FUNCTION_BLOCK UN_CleanroomConnect EXTENDS Un_Base
VAR
//------------------------------------------//
//Function Blocks

//------------------------------------------//



//------------------------------------------//
//Control Modules (Devices)
	s_CmKmweLeds 				: CM_KmweLeds;
//------------------------------------------//

//------------------------------------------//
//Inputs
	s_diEmergencyBtn			: FB_DigInput;
//------------------------------------------//

//------------------------------------------//
//Alarms
	s_errEmergencyBtn			: FB_AlarmHandler;
//------------------------------------------//
	
//------------------------------------------//
//Params

//------------------------------------------//

//------------------------------------------//
//Variables
	s_stSqldbSettings			: ST_SqLdbConfiguration;
//------------------------------------------//

//------------------------------------------//
//Properties

//------------------------------------------//

//------------------------------------------//
//Hmi
	s_fbHmiBtnAutomatic			: FB_HmiBtn;
	s_fbHmiBtnManual			: FB_HmiBtn;
	s_fbHmiBtnTesterConfig		: FB_HmiBtn;
	s_fbHmiBtnAlarms			: FB_HmiBtn;
//------------------------------------------//
END_VAR


SUPER^();

METHOD PROTECTED _m_Alarms : BOOL

IF NOT SUPER^._m_Alarms() THEN
	RETURN;
END_IF

//overbruggen in automode tot en met place table blablabla
s_errEmergencyBtn(i_bStaActive 			:= NOT s_DiEmergencyBtn.p_bStaInput AND NOT GVL.g_fbHmiBtnSimulation.p_bStaBtn AND GVL.g_bConnectTestEquipment ,
				  i_eAlarmLevel 		:= E_AlarmLevel.Alarm,
				  i_sAlarmText 			:= 'Emergency button pressed');

IF GVL_KMWEGenericLib.g_fbAlarmManager.p_bAlarmActive THEN 
	GVL.g_eStaLedColor := E_KmweLedColors.Red;
END_IF

s_bStaError := s_errEmergencyBtn.q_bStaActive;

_m_Alarms := TRUE;
END_METHOD

METHOD PROTECTED _m_Devices : BOOL

IF NOT SUPER^._m_Devices() THEN
	RETURN;
END_IF

//------------------------------------------//
//CM
	s_CmKmweLeds(i_bReqEnable := TRUE,
			 i_bCmdReset  := s_bCmdReset,
			 i_eCtrlMode  := s_eCtrlMode,
			 i_eColor 	  := GVL.g_eStaLedColor);
			 
	s_CmKmweLeds.p_bFlashFast := GVL.g_bLedFlashFast;
	s_CmKmweLeds.p_bFlashSlow := GVL.g_bLedFlashSlow;

//------------------------------------------//

//------------------------------------------//
//Outputs
//------------------------------------------//

//------------------------------------------//
//Inputs
	s_diEmergencyBtn();	
//------------------------------------------//

_m_Devices := TRUE;
END_METHOD

METHOD PROTECTED _m_Hmi : BOOL
VAR_INST
	s_sPrevPageAlarms 		: STRING;
	s_sPrevBottom1Alarms	: STRING;
	
	s_sCompanySelectionVisible	: STRING;
END_VAR

IF NOT SUPER^._m_Hmi() THEN
	RETURN;
END_IF

//------------------------------------------//
//Mode management
IF GVL_KMWEGenericLib.g_fbHmiBtnReturnToStart.p_osfBtnPress THEN
	s_eCtrlMode := E_CtrlMode.IDLE;

	GVL_KMWEGenericLib.g_fbHmiBtnAcknowledge.p_bStaVisible	:= TRUE;
	GVL_KMWEGenericLib.g_fbHmiBtnAcknowledge.p_bStaEnabled	:= TRUE;	
END_IF
//------------------------------------------//

//------------------------------------------//
//Alarm Button can always be pressed
IF s_fbHmiBtnAlarms.p_osrBtnPress AND GVL.g_sToHmiMiddleContent <> GVL.g_stHmiMiddle.AlarmManager THEN
	s_sPrevPageAlarms			:= GVL.g_sToHmiMiddleContent;
	s_sPrevBottom1Alarms		:= GvL.g_sToHmiBottomContent;
	GVL.g_sToHmiMiddleContent 	:= GVL.g_stHmiMiddle.AlarmManager;
	GVL.g_sToHmiBottomContent	:= GVL.g_stHmiBottomBar.Alarm;
	
	GVL_KMWEGenericLib.g_fbHmiBtnReturn.p_bStaVisible 			:= TRUE;
	GVL_KMWEGenericLib.g_fbHmiBtnReturn.p_bStaEnabled 			:= TRUE;
END_IF

IF GVL.g_sToHmiMiddleContent = GVL.g_stHmiMiddle.AlarmManager AND GVL_KMWEGenericLib.g_fbHmiBtnReturn.p_osfBtnPress THEN
	GVL.g_sToHmiMiddleContent 	:=	s_sPrevPageAlarms;
	GVL.g_sToHmiBottomContent	:=	s_sPrevBottom1Alarms;
	
	GVL_KMWEGenericLib.g_fbHmiBtnReturn.p_bStaVisible 			:= FALSE;
	GVL_KMWEGenericLib.g_fbHmiBtnReturn.p_bStaEnabled 			:= FALSE;
END_IF
//------------------------------------------//

//------------------------------------------//
//Hmi view management (General, Em can set module specific pages)
CASE s_eCtrlMode OF
	E_CtrlMode.IDLE:
		GVL.g_bConnectTestEquipment		:= TRUE;

		IF NOT GVL_KMWEGenericLib.g_fbAlarmManager.p_bAlarmActive THEN
			GVL.g_bLedFlashFast	:= FALSE;
			GVL.g_bLedFlashSlow	:= FALSE;
			GVL.g_eStaLedColor := E_KmweLedColors.Idle;
		END_IF
	
		s_fbHmiBtnTesterConfig.p_sBtnText		:= 'Tester Configuration';	
	
		IF GVL_KMWEGenericLib.g_fbHmiBtnReturnToStart.p_osfBtnPress THEN
			GVL_KMWEGenericLib.g_fbParamManager.p_bShowHmiParam := FALSE;

			GVL.g_sToHmiMiddleContent 	:= GVL.g_stHmiMiddle.Start;
			GVL.g_sToHmiBottomContent	:= GVL.g_stHmiBottomBar.Start;
		END_IF
		
		IF s_fbHmiBtnTesterConfig.p_osrBtnPress THEN
			GVL_KMWEGenericLib.g_fbParamManager.p_nFolderIndex 	:= 1;
			GVL_KMWEGenericLib.g_fbParamManager.p_bShowHmiParam := TRUE;

			GVL.g_sToHmiMiddleContent 	:= GVL.g_stHmiMiddle.TesterConfig;
			GVL.g_sToHmiBottomContent	:= GVL.g_stHmiBottomBar.General_ReturnToStart;
		END_IF
		
		IF s_fbHmiBtnAutomatic.p_osrBtnPress THEN
			s_eCtrlMode 					:= E_CtrlMode.AUTOMATIC;
			GVL.g_bConnectTestEquipment		:= FALSE;
			
			GVL_KMWEGenericLib.g_fbHmiBtnAcknowledge.p_sBtnText		:= 'Acknowledge';
			
			GVL_KMWEGenericLib.g_fbParamManager.p_nFolderIndex 		:= 2;
			
			GVL_KMWEGenericLib.g_fbHmiBtnAcknowledge.p_bStaVisible	:= FALSE;
			GVL_KMWEGenericLib.g_fbHmiBtnAcknowledge.p_bStaEnabled	:= FALSE;
	
			GVL_KMWEGenericLib.g_fbHmiBtnReturn.p_bStaVisible		:= TRUE;
			GVL_KMWEGenericLib.g_fbHmiBtnReturn.p_bStaEnabled		:= TRUE;
			
			GVL.g_sToHmiMiddleContent 	:= GVL.g_stHmiMiddle.OperatorInputData;
			GVL.g_sToHmiBottomContent	:= GVL.g_stHmiBottomBar.Procedure;
		END_IF
		
		IF s_fbHmiBtnManual.p_osrBtnPress THEN
			s_eCtrlMode := E_CtrlMode.MANUAL;
			
			GVL.g_sToHmiMiddleContent 	:= GVL.g_stHmiMiddle.Manual;
			GVL.g_sToHmiBottomContent	:= GVL.g_stHmiBottomBar.General_ReturnToStart;
		END_IF

	E_CtrlMode.AUTOMATIC:
		s_fbHmiBtnTesterConfig.p_sBtnText		:= 'Procedure Configuration';
		
		IF GVL.g_sToHmiMiddleContent = GVL.g_stHmiMiddle.OperatorInputData 
			AND GVL_KMWEGenericLib.g_fbHmiBtnReturn.p_osrBtnPress 
		THEN
			GVL_KMWEGenericLib.g_fbParamManager.p_bShowHmiParam := FALSE;

			GVL.g_sToHmiMiddleContent 							:= GVL.g_stHmiMiddle.Start;
			GVL.g_sToHmiBottomContent							:= GVL.g_stHmiBottomBar.Start;
			
			s_eCtrlMode 										:= E_CtrlMode.IDLE;	
		END_IF
		
		IF s_fbHmiBtnTesterConfig.p_osrBtnPress THEN
			GVL_KMWEGenericLib.g_fbParamManager.p_nFolderIndex 	:= 2;
			GVL_KMWEGenericLib.g_fbParamManager.p_bShowHmiParam := TRUE;

			GVL_KMWEGenericLib.g_fbHmiBtnAcknowledge.p_bStaVisible	:= FALSE;
			GVL_KMWEGenericLib.g_fbHmiBtnAcknowledge.p_bStaEnabled	:= FALSE;
			
			GVL_KMWEGenericLib.g_fbHmiBtnReturn.p_bStaVisible		:= TRUE;
			GVL_KMWEGenericLib.g_fbHmiBtnReturn.p_bStaEnabled		:= TRUE;

			GVL.g_sToHmiMiddleContent 	:= GVL.g_stHmiMiddle.TesterConfig;
			GVL.g_sToHmiBottomContent	:= GVL.g_stHmiBottomBar.General_Return;
		END_IF
		
		IF GVL.g_sToHmiMiddleContent = GVL.g_stHmiMiddle.TesterConfig THEN
			IF GVL_KMWEGenericLib.g_fbHmiBtnReturn.p_osrBtnPress THEN
				GVL.g_sToHmiMiddleContent 	:= GVL.g_stHmiMiddle.OperatorInputData;
				GVL.g_sToHmiBottomContent	:= GVL.g_stHmiBottomBar.Procedure;
				
				GVL_KMWEGenericLib.g_fbHmiBtnReturn.p_bStaVisible		:= FALSE;
				GVL_KMWEGenericLib.g_fbHmiBtnReturn.p_bStaEnabled		:= FALSE;
			END_IF
		END_IF
		
	E_CtrlMode.MANUAL:
		IF GVL_KMWEGenericLib.g_fbAlarmManager.p_osrAlarmsResolved THEN
			GVL.g_eStaLedColor := E_KmweLedColors.Green;
		END_IF
	
		GVL_KMWEGenericLib.g_fbHmiBtnAcknowledge.p_bStaVisible	:= FALSE;
		GVL_KMWEGenericLib.g_fbHmiBtnAcknowledge.p_bStaEnabled	:= FALSE;
		
//		IF GVL_KMWEGenericLib.g_fbHmiBtnReturnToStart.p_osrBtnPress THEN
//			GVL.g_sToHmiMiddleContent 	:= ST_HmiMiddle.Start;
//			GVL.g_sToHmiBottomContect	:= ST_HmiBottomBar.Start;
//		END_IF
		;
END_CASE
//------------------------------------------//

//------------------------------------------//
//Hmi Buttons
s_fbHmiBtnAutomatic();
s_fbHmiBtnManual();
s_fbHmiBtnTesterConfig();
s_fbHmiBtnAlarms();
GVL.g_fbHmiBtnSimulation();
//------------------------------------------//
END_METHOD

METHOD PROTECTED _m_Init : BOOL

IF NOT SUPER^._m_Init() THEN
	RETURN;
END_IF

_m_AddModule(i_itfModuleBase := GVL_Modules.g_EmRMMTTester);

//------------------------------------------//
//Hmi Startup
GVL.g_sToHmiTopContent 		:= GVL.g_stHmiTopBar.GeneralTopbar;
GVL.g_sToHmiMiddleContent 	:= GVL.g_stHmiMiddle.Start;
GVL.g_sToHmiBottomContent	:= GVL.g_stHmiBottomBar.Start;
//------------------------------------------//

//------------------------------------------//
//Buttons
	s_fbHmiBtnAutomatic.p_bStaEnabled 		:= TRUE;
	s_fbHmiBtnAutomatic.p_bStaVisible 		:= TRUE;
	s_fbHmiBtnAutomatic.p_eButtontype		:= E_HmiButtonType.PUSHBUTTON;
	s_fbHmiBtnAutomatic.p_sBtnText			:= 'Auto';

	s_fbHmiBtnManual.p_bStaEnabled 			:= TRUE;
	s_fbHmiBtnManual.p_bStaVisible 			:= TRUE;
	s_fbHmiBtnManual.p_eButtontype			:= E_HmiButtonType.PUSHBUTTON;
	s_fbHmiBtnManual.p_sBtnText				:= 'Manual';
	
	s_fbHmiBtnTesterConfig.p_bStaEnabled 	:= TRUE;
	s_fbHmiBtnTesterConfig.p_bStaVisible 	:= TRUE;
	s_fbHmiBtnTesterConfig.p_eButtontype	:= E_HmiButtonType.PUSHBUTTON;
	s_fbHmiBtnTesterConfig.p_sBtnText		:= 'Configuration';
	
	s_fbHmiBtnAlarms.p_bStaVisible 			:= TRUE;
	s_fbHmiBtnAlarms.p_bStaEnabled			:= TRUE;
	s_fbHmiBtnAlarms.p_eButtontype 			:= E_HmiButtonType.PUSHBUTTON;
	s_fbHmiBtnAlarms.p_sBtnText				:= 'Alarms';

	GVL.g_fbHmiBtnSimulation.p_bStaVisible 	:= TRUE;
	GVL.g_fbHmiBtnSimulation.p_bStaEnabled	:= TRUE;
	GVL.g_fbHmiBtnSimulation.p_eButtontype 	:= E_HmiButtonType.TOGGLEBUTTON;
	GVL.g_fbHmiBtnSimulation.p_sBtnText		:= 'Simulation';
	
	GVL_KMWEGenericLib.g_fbHmiBtnReturn.p_bStaVisible 	:= FALSE;
	GVL_KMWEGenericLib.g_fbHmiBtnReturn.p_bStaEnabled 	:= FALSE;
//------------------------------------------//


//------------------------------------------//
//Database information
s_stSqldbSettings.sServer				:= 'plc-db\sqlexpress';
s_stSqldbSettings.sProvider				:= 'SQLOLEDB';
s_stSqldbSettings.sDatabase				:= 'RMMT_Tester';
s_stSqldbSettings.sUserID				:= 'RMMT_Tester';
s_stSqldbSettings.sPassword				:= 'dCH9FTVALtsukUQMv5yjWr';
s_stSqldbSettings.bAuthentification		:= TRUE;
//------------------------------------------//

_m_Init := TRUE;
END_METHOD

METHOD PROTECTED _m_Modules : BOOL

//Interlocks (TRUE = interlocked)
GVL_Modules.g_emDoors.i_bIlckOuterDoorToClose := 
	GVL_Modules.g_emDockingInterface.p_bStaDockingDone;
	
GVL_Modules.g_emDoors.i_bIlckOuterDoorToOpen :=
	NOT(GVL_Modules.g_emDoors.p_bStaCleanroomDoorClosed)
	OR NOT(GVL_Modules.g_emDoors.p_bStaCleanroomLockApplied);
//++	OR NOT(GVL_Modules.emAirTreathment.p_bStaRunningOk;
 
GVL_Modules.g_emDoors.i_bIlckCleanroomDoorToLock := 
	NOT(GVL_Modules.g_emDoors.p_bStaCleanroomDoorClosed);

GVL_Modules.g_emDoors.i_bIlckCleanroomDoorToRelease :=
	( NOT(GVL_Modules.g_emDoors.p_bStaOuterDoorClosed) AND NOT(GVL_Modules.g_emDockingInterface.p_bStaDockingDone) );
	//++	OR NOT(GVL_Modules.emAirTreathment.p_bStaRunningOk;

GVL_Modules.g_emStateMachine(
	i_bReqEnable := TRUE,
	i_eCtrlMode := s_eCtrlMode,
	i_bCmdReset := p_bCmdReset,
	i_sEmName := 'EM State Machine',
	i_itfEmDoors := GVL_Modules.g_emDoors,
	i_itfEmDockingInterface := GVL_Modules.g_emDockingInterface);

GVL_Modules.g_emDoors(
	i_bReqEnable := TRUE,
	i_eCtrlMode := s_eCtrlMode,
	i_bCmdReset := p_bCmdReset,
	i_sEmName := 'EM Doors');

GVL_Modules.g_emDockingInterface(
	i_bReqEnable := TRUE,
	i_eCtrlMode := s_eCtrlMode,
	i_bCmdReset := p_bCmdReset,
	i_sEmName := 'EM Docking Interface');
	
//++GVL_Modules.g_emAirTreatment(
//++	i_bReqEnable := TRUE,
//++	i_eCtrlMode := s_eCtrlMode,
//++	i_bCmdReset := p_bCmdReset,
//++	i_sEmName := 'EM Air Treatment');	
	
s_bStaError :=
	GVL_Modules.g_emDoors.q_bStaError
	OR GVL_Modules.g_emDockingInterface.q_bStaError;
//++	OR GVL_Modules.g_emAirTreatment.q_bStaError;
	
_m_Modules := TRUE;
END_METHOD

METHOD PRIVATE _m_SelectConfigFile : BOOL
VAR_INPUT
	i_bCmdReset 			: BOOL;
END_VAR
VAR_INST	
	i, x					: UDINT;
		
	s_aPossibleRevs			: ARRAY[0..TO_DINT(Param_Project.n_MaxParamFiles)] OF T_MAXSTRING;
	
	s_aConfigFileNames 		: ARRAY[0..Param_Project.n_MaxParamFiles] OF T_MAXSTRING;
	s_aConfigFileDUTs		: ARRAY[0..TO_DINT(Param_Project.n_MaxParamFiles)] OF T_MAXSTRING;	
	s_aConfigFileRev		: ARRAY[0..Param_Project.n_MaxParamFiles] OF T_MAXSTRING;
	
	s_aSingleDUTs			: ARRAY[0..TO_DINT(Param_Project.n_MaxParamFiles)] OF T_MAXSTRING;
	s_aSingleREVs			: ARRAY[0..TO_DINT(Param_Project.n_MaxParamFiles)] OF T_MAXSTRING;
		
	s_nIndexDut				: INT;
//	s_nIndexSR				: INT;
	s_nIndexRev				: INT;
	
	s_nIndexDutPrev			: INT;
	s_nIndexRevPrev			: INT;
	
	s_sChosenFile			: T_MAXSTRING;
	s_sToHmiChosenFile		: T_MAXSTRING;
	
	s_bCmdResetInternal	 	: BOOL;
END_VAR

//1413824/E test bestand met deze naam.

IF i_bCmdReset OR s_bCmdResetInternal THEN	
	MEMSET(ADR(s_aConfigFileNames), 0, SIZEOF(s_aConfigFileNames));
	MEMSET(ADR(s_aConfigFileDUTs), 0, SIZEOF(s_aConfigFileDUTs));
	MEMSET(ADR(s_aSingleDUTs), 0, SIZEOF(s_aSingleDUTs));
	
	MEMCPY(ADR(s_aConfigFileNames), ADR(GVL_KMWEGenericLib.g_fbParamManager.s_aFileListHmi), SIZEOF(GVL_KMWEGenericLib.g_fbParamManager.s_aFileListHmi));
	
	s_nIndexDut		:= -1;
//	s_nIndexSR		:= -1;
	s_nIndexRev		:= -1;
	
	FOR i := 0 TO Param_Project.n_MaxParamFiles DO 
		FindAndSplit(pSeparator:= ADR('^'),
							 pSrcString:= ADR(s_aConfigFileNames[i]),
							 pLeftString:= ADR(s_aConfigFileDUTs[i]),
							 nLeftSize:= SIZEOF(s_aConfigFileDUTs[i]),
							 pRightString:= ADR(s_aConfigFileRev[i]),
							 nRightSize:= SIZEOF(s_aConfigFileRev[i]),
							 bSearchFromRight:= FALSE);	

		s_aConfigFileRev[i] := 	DELETE(s_aConfigFileRev[i], 6, 2);			
	END_FOR
	
	F_CheckDuplicatesInArray(iq_aOriginalArray := s_aConfigFileDUTs, iq_aUniqueArray := s_aSingleDUTs);

	IF s_aConfigFileNames[0] = '' THEN
		s_bCmdResetInternal := TRUE;	
	ELSE
		s_bCmdResetInternal := FALSE;	
	END_IF
END_IF

IF s_nIndexDutPrev <> s_nIndexDut AND s_nIndexDutPrev <> -1 THEN
	s_nIndexRev := -1;
	
	MEMSET(ADR(s_aSingleREVs), 0, SIZEOF(s_aSingleREVs));
END_IF

IF s_nIndexDut <> -1 AND s_nIndexRev = -1 THEN 
	x := 0;
	MEMSET(ADR(s_aSingleREVs), 0, SIZEOF(s_aSingleREVs));
	MEMSET(ADR(s_aPossibleRevs), 0, SIZEOF(s_aPossibleRevs));
	FOR i:= 0 TO Param_Project.n_MaxParamFiles DO
		IF FIND(s_aConfigFileNames[i], s_aSingleDUTs[s_nIndexDut]) <> 0 THEN
			s_aPossibleRevs[x] := MID(s_aConfigFileNames[i],1,FIND(s_aConfigFileNames[i], '^')+1);
			x := x + 1;
		END_IF					
	END_FOR	
	
	F_CheckDuplicatesInArray(iq_aOriginalArray := s_aPossibleRevs, iq_aUniqueArray := s_aSingleREVs); 
END_IF

IF s_nIndexDut <> -1 AND s_nIndexRev <> -1 AND s_nIndexRevPrev <> s_nIndexRev THEN
	FOR i := 0 TO Param_Project.n_MaxParamFiles DO
		IF s_aConfigFileNames[i] = CONCAT(s_aSingleDUTs[s_nIndexDut], 
										CONCAT('^', 
										CONCAT(s_aSingleRevs[s_nIndexRev], '.csv')))
		THEN
			s_sChosenFile := s_aConfigFileNames[i];
		END_IF
	END_FOR
	
	FOR i := 0 TO Param_Project.n_MaxParamFiles DO
		IF GVL_KMWEGenericLib.g_fbParamManager.s_aFileListHmi[i] = s_sChosenFile THEN
			GVL_KMWEGenericLib.g_fbParamManager.p_nHmiFileSelected := TO_UDINT(i);
		END_IF
	END_FOR 
END_IF

IF s_aConfigFileNames[GVL_KMWEGenericLib.g_fbParamManager.p_nHmiFileSelected] <> s_sChosenFile THEN
	s_nIndexDut	:= -1;
	s_nIndexRev	:= -1;
	
	MEMSET(ADR(s_aSingleREVs), 0, SIZEOF(s_aSingleREVs));
END_IF

s_sChosenFile 		:= GVL_KMWEGenericLib.g_fbParamManager.s_aFileListHmi[GVL_KMWEGenericLib.g_fbParamManager.p_nHmiFileSelected];
s_sToHmiChosenFile 	:= DELETE(s_sChosenFile, 4, FIND(s_sChosenFile, '.csv'));

s_nIndexRevPrev := s_nIndexRev;
s_nIndexDutPrev	:= s_nIndexDut;
END_METHOD

METHOD PUBLIC m_FastTask : BOOL

CASE GVL_DataLogging.g_eDataAction OF
	E_DataReadWriteActions.MagneticProcedure:
			GVL_DataLogging.g_fbDataLogger.m_FastTask(iq_aCSVFieldFast 			:= GVL_Datalogging.g_aLoggingDataMagnetic,
														i_bCmdResetReadFast 	:= GVL_Datalogging.g_bCmdResetReadFast,
														i_bCmdResetWriteFast 	:= GVL_Datalogging.g_bCmdResetWriteFast,
														i_sFileName 			:= GVL_Datalogging.g_sFilenameFast);				
END_CASE
END_METHOD

METHOD PUBLIC m_Main : BOOL

IF NOT SUPER^.m_Main() THEN
	RETURN;
END_IF

GVL.g_osrNotify();

//--GVL_DataLogging.g_fbDataLogger(i_sPathName := 'C:\RMMT\', i_bCmdReset := s_bCmdReset);

//--GVL_DataLogging.g_fbSqlDatabase(i_stSettings := s_stSqlDbSettings, i_bCmdReset := s_bCmdReset);

//--_m_SelectConfigFile(i_bCmdReset := s_fbHmiBtnAutomatic.p_osfBtnPress);

GVL.g_osrNotify.CLK := FALSE;	

m_Main := TRUE;



// Paul Schippers: just a test with the use of interfaces
itfEmDoors.m_CloseOuterDoor();

itfEmDockingInterface.m_OpenDockingClamps();

//IF NOT(itfEmAirTreatment.p_bStaPressurizingOK) THEN 
//	itfEmAirTreatment.m_Pressurize();
//END_IF

(*	
	// Interlocks (doors must work as an airlock, only one door may be opened at all times)
	s_bIlckSpeedDoorOuterToOpen :=
		s_cmDoorLockCleanroom.p_bStaError
		OR NOT(s_cmDoorLockCleanroom.p_bStaEnabled)
		NOT(s_cmDoorLockCleanroom.p_bStaDoorIsClosed)
		OR NOT (s_cmDoorLockCleanroom.p_bStaLockIsApplied)
		OR s_cmDoorLockCleanroom.p_bStaLockIsReleased
		OR TRUE (*Air treathment unit must be running and ok*)
		OR TRUE (*Add more..*);
	s_bIlckSpeedDoorOuterToClose :=
		TRUE (*Opening must be free*)
		OR TRUE (*Add more..*);
	
	s_bIlckDoorLockCleanroomToOpen :=
		s_cmSpeedDoorOuter.p_bStaError
		OR NOT(s_cmSpeedDoorOuter.p_bStaEnabled)
		OR NOT(s_cmSpeedDoorOuter.p_bStaIsClosed)
		OR s_cmSpeedDoorOuter.p_bStaIsClosing
		OR s_cmSpeedDoorOuter.p_bStaIsOpened
		OR s_cmSpeedDoorOuter.p_bStaIsOpening
		OR TRUE (*Air treathment unit must be running and ok*)
		OR TRUE (*Add more..*);
*)
END_METHOD

END_FUNCTION_BLOCK

(* stored: Version 1.1.0.1, ProductVersion 3.1.4024.12
   POU UN_CleanroomConnect: Id {8b93890b-f796-4713-9491-f75e01fbeba7}, SpecialFunc None
   Method _m_Alarms: Id {c0f56159-8f50-4d36-acac-c259038873b1}
   Method _m_Devices: Id {68eeb98b-de01-4c23-9e4b-e0a75e4ed7ba}
   Method _m_Hmi: Id {6e489294-edbd-4c11-9b41-7f97eb3787da}
   Method _m_Init: Id {71192b96-a840-4eae-8166-473534974241}
   Method _m_Modules: Id {2372c80a-8810-4c92-8500-979916e08046}
   Method _m_SelectConfigFile: Id {7c7e81b7-08ef-4473-8a6d-b20d88aaf565}
   Method m_FastTask: Id {d7f04e67-2f14-466a-aab3-c133442def96}
   Method m_Main: Id {bf5d9d9d-3881-4722-ad23-ed0781ff35d5} *)
